# B&R Automation Studio project FileHandling
Automation Studio 4.9

## Configuration Config1

CPU X20CP0484, AutomationRuntime 6.0.2, Build 11.3.0, Vc 6.0.0

### Task classes (Cpu.sw)
```
Cyclic#4 (cycle 100000 us, tolerance 100000 us):
  fileHandli <- fileHandling.prg
Libraries: runtime, standard
```

### Hardware
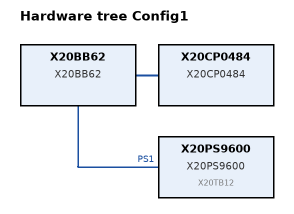
```
X20BB62 : X20BB62 v1.3.0.0
X20CP0484 : X20CP0484 v1.8.1.0  [SL -> X20BB62.SL1]
  Connector IF2:
    ActivateDevice = 1
    ActivateSnmp = 2
  Connector IF3:
    CycleTime = 400
  ConfigurationID = FileHandling_Config1
  Simulation = 1
  TimerDeviceType = SWIOTIMER
  Cyclic1Duration = 10000
  Cyclic1Tolerance = 10000
  Cyclic2Duration = 20000
  Cyclic2Tolerance = 20000
  Cyclic3Duration = 50000
  Cyclic3Tolerance = 50000
  Cyclic4Duration = 100000
  Cyclic4Tolerance = 100000
  Cyclic5Duration = 200000
  Cyclic5Tolerance = 200000
  Cyclic6Duration = 500000
  Cyclic6Tolerance = 500000
  Cyclic7Duration = 1000000
  Cyclic7Tolerance = 1000000
  Cyclic8Duration = 10000
  Cyclic8Tolerance = 30000000
  FileDevice1
  FileDeviceName1 = USER
  FileDevicePath1 = USER_PATH
  FileDevice2
  FileDeviceName2 = F
  FileDevicePath2 = F:
  FileDevice3
  FileDeviceName3 = TEST
  FileDevicePath3 = F:/test
  FileDevice4
  FileDeviceName4 = C
  FileDevicePath4 = C:
  FileDevice5
  FileDeviceName5 = D
  FileDevicePath5 = D:
  ActivateFtpServer = 1
  FTPProtocol = 1
  FtpUser1
  FtpUsername1 = admin
  FtpUserPassword1 = nIM63jTojMQbPoAbPMbmFY5hcHAc9f+6nMOFN6eV5vc=  // admin
  FtpUserSalt1 = sRD2ml1v
  FTPAccessRight1 = 0
  FTPdevice1 = ALL
X20PS9600 : X20PS9600 v1.6.2.0  [PS -> X20BB62.PS1; SS1 -> X20TB12.SS]
X20TB12 : X20TB12 v1.0.0.0
```

## Logical view

Binary libraries used (declarations not repeated): operator, runtime, AsIecCon, astime, FileIO, standard


### Program Logical/fileHandling (IEC)

#### Variables.var
```iecst
VAR
	FileOpen_0 : FileOpen;
	FileRead_0 : FileRead;
	FileWrite_0 : FileWrite;
	FileClose_0 : FileClose;
	FileCreate_0 : FileCreate;
	FileDelete_0 : FileDelete;
	DirInfo_0 : DirInfo;
	DirRead_0 : DirRead;
	DirCreate_0 : DirCreate;
	data : STRING[80];
	fileName : STRING[80];
	ident : UDINT;
	state : USINT;
	writeFile : BOOL;
	readFile : BOOL;
	deleteFile : BOOL;
	clear : BOOL;
	dirName : STRING[80];
	deviceName : STRING[80];
END_VAR
```

#### Main.st
```iecst
PROGRAM _INIT
	(* Insert code here *)
	data := 'Hello, I am some data that would like to be written to a file';
	fileName := 'testFile.txt';
END_PROGRAM

PROGRAM _CYCLIC
	(* Insert code here *)

	CASE state OF
		0:
			// base case
			// waiting for command
			IF writeFile THEN
				writeFile := FALSE;
				state := 10;
			END_IF

			IF readFile THEN
				readFile := FALSE;
				state := 40;
			END_IF

			IF deleteFile THEN
				deleteFile := FALSE;
				state := 70;
			END_IF

		10:
			// open file
			FileOpen_0.enable 	:= TRUE;
			FileOpen_0.pDevice 	:= ADR('F');
			FileOpen_0.pFile 	:= ADR(fileName);
			FileOpen_0.mode 	:= fiREAD_WRITE;
			state := 15;

		15:
			// wait for response
			ident := FileOpen_0.ident;
			IF FileOpen_0.status = fiERR_FILE_NOT_FOUND THEN
				FileOpen_0.enable := FALSE;
				state := 20;
			ELSIF FileOpen_0.status = ERR_FUB_BUSY THEN
				// wait
			ELSIF FileOpen_0.status = ERR_OK THEN
				FileOpen_0.enable := FALSE;
				state := 30;
			ELSE // error
				FileOpen_0.enable := FALSE;
				state := 99;
			END_IF

		20:
			// create file
			FileCreate_0.enable		:= TRUE;
			FileCreate_0.pDevice 	:= ADR('F');
			FileCreate_0.pFile 		:= ADR(fileName);
			state := 25;

		25:
			// wait for creating
			ident := FileCreate_0.ident;
			IF FileCreate_0.status = ERR_FUB_BUSY THEN
				// wait
			ELSIF FileCreate_0.status = ERR_OK THEN
				FileCreate_0.enable	:= FALSE;
				state := 30;
			ELSE // error
				FileCreate_0.enable	:= FALSE;
				state := 99;
			END_IF

		30:
			// write file
			FileWrite_0.enable := TRUE;
			FileWrite_0.ident := ident;
			FileWrite_0.pSrc := ADR(data);
			FileWrite_0.len := LEN(data); // could also be SIZEOF depending on the datatype
			state := 35;

		35:
			// waiting for writing
			IF FileWrite_0.status = ERR_FUB_BUSY THEN
				// wait
			ELSIF FileWrite_0.status = ERR_OK THEN
				FileWrite_0.enable := FALSE;
				state := 60;
			ELSE
				FileWrite_0.enable := FALSE;
				state := 99;
			END_IF

		40:
			// read file
			// open file
			FileOpen_0.enable 	:= TRUE;
			FileOpen_0.pDevice 	:= ADR('F');
			FileOpen_0.pFile 	:= ADR(fileName);
			FileOpen_0.mode 	:= fiREAD_ONLY;
			state := 45;

		45:
			// wait for response
			ident := FileOpen_0.ident;
			IF FileOpen_0.status = fiERR_FILE_NOT_FOUND THEN
				FileOpen_0.enable := FALSE;
				state := 99;
			ELSIF FileOpen_0.status = ERR_FUB_BUSY THEN
				// wait
			ELSIF FileOpen_0.status = ERR_OK THEN
				state := 50;
			ELSE // error
				FileOpen_0.enable := FALSE;
				state := 99;
			END_IF

		50:
			FileRead_0.enable 	:= TRUE;
			FileRead_0.ident 	:= ident;
			FileRead_0.len 		:= FileOpen_0.filelen;
			FileRead_0.pDest 	:= ADR(data);
			state := 60;

		60:
			// close file
			FileClose_0.enable 	:= TRUE;
			FileClose_0.ident 	:= ident;
			state := 65;

		65:
			IF FileClose_0.status = ERR_FUB_BUSY THEN
				// wait
			ELSIF FileClose_0.status = ERR_OK THEN
				FileClose_0.enable := FALSE;
				state := 0;
			ELSE
				state := 99;
			END_IF

		70:
			// delete file
			FileDelete_0.enable 	:= TRUE;
			FileDelete_0.pDevice 	:= ADR('F');
			FileDelete_0.pName 		:= ADR(fileName);
			state := 75;

		75:
			IF FileDelete_0.status = ERR_FUB_BUSY THEN
				// wait
			ELSIF FileDelete_0.status = ERR_OK THEN
				FileDelete_0.enable := FALSE;
				state := 0;
			ELSE
				state := 99;
			END_IF

		99:
		// error
			IF clear THEN
				clear 				:= FALSE;
				FileOpen_0.enable 	:= FALSE;
				FileCreate_0.enable := FALSE;
				FileWrite_0.enable 	:= FALSE;
				FileRead_0.enable 	:= FALSE;
				FileClose_0.enable 	:= FALSE;
				FileDelete_0.enable := FALSE;
			END_IF
	END_CASE

	FileOpen_0();
	FileCreate_0();
	FileWrite_0();
	FileRead_0();
	FileClose_0();
	FileDelete_0();

	DirInfo_0.pDevice := ADR(deviceName);
	DirInfo_0.pPath := ADR(dirName);
	DirInfo_0();

END_PROGRAM

PROGRAM _EXIT
	(* Insert code here *)

END_PROGRAM
```

Listed in the project but not available here: Logical/Global.typ, Logical/Global.var
